TYPE M3TranslationGotoArgs :
STRUCT
	///Position setpoint of the translation stage, in millimeters
	position: LREAL;
END_STRUCT
END_TYPE

(* stored: Version 1.1.0.1, ProductVersion 3.1.4019.2
   DUT M3TranslationGotoArgs: Id {ed933b0c-7fe5-4ce8-9aac-84c77088823e} *)
